PROGRAM MAIN
VAR
	rtStep						:R_Trig;
	
	rtAck						:R_Trig;
	i							:UDINT;
	fbWakeUpTmr					:TON;	
	sTime						:STRING(8);
	bAckLED						:BOOL;
	darius						:UDINT;	
	
	// Alarm	
	aErrorActive				:ARRAY[1..nNbrOfAlarms] OF WORD;
	aErrorID1					:ARRAY[1..nNbrOfAlarms] OF STRING(255);
	aErrorID2					:ARRAY[1..nNbrOfAlarms] OF STRING(255);
	afbAlarms					:ARRAY[1..nNbrOfAlarms] OF FB_TcAlarm;
	fbSource					:FB_TcSourceInfo;

	(*Vise station components*)
	rtStepViseStation			:R_Trig;

END_VAR

//InitTCPIP();
Init();
Blink();
SafetyPRG();
Alarm();
BusDiag();
Door();
Light();
Mode();
ViseProgram();
RobotCncProgram();
Robot7AxisProgram();
CNC_1();
CNC_3();
ConveyorSystem();
Mapping();

Test();
SQL_Test();


fbTime(bEnable := TRUE, dwCycle := 1);
dtSystemTime := SYSTEMTIME_TO_DT(TIMESTR:= fbTime.systemTime);
sTime := MID((SYSTEMTIME_TO_STRING(fbTime.systemTime)),8,12);

ACTION Alarm:
// Creating error acknowladge impulse
rtAck(CLK:= i_bVisePos1ErrorAckBtn OR i_bVisePos2ErrorAckBtn OR bAckHMI OR i_bErrorAckBtn_Main, Q=> bAckP);
IF rtAck.Q THEN
	afbAlarms[1].Confirm(0); afbAlarms[2].Confirm(0); afbAlarms[3].Confirm(0); afbAlarms[4].Confirm(0);
	afbAlarms[5].Confirm(0); afbAlarms[6].Confirm(0); afbAlarms[7].Confirm(0); 
	bAckHMI := FALSE;
END_IF

IF wError <> 0 OR bSafetyError_CNC45 OR ViseProgram.nState >= 200000 THEN
	bGlobalError := TRUE;
ELSE
	bGlobalError := FALSE;
END_IF

(* 
	wError.0 : Air pressure error
	wError.1 : Ethercat error
	wError.2 : 
	wError.3 : 
	wError.4 : 
	wError.5 : 
	wError.6 : 
	wError.7 : 
	wError.8 : 
	wError.9 : 
*)

aErrorActive[1].0 := wError.0;
aErrorActive[2].0 := wError.1;
aErrorActive[3].0 := i_bSafetyGroupComErr_CNC45;
aErrorActive[4].0 := i_bSafetyGroupFBErr_CNC45;
aErrorActive[5].0 := i_bSafetyGroupOtherErr_CNC45;
aErrorActive[6].0 := i_bLO1EDMErr_CNC45;
aErrorActive[7].0 := i_bLO2EDMErr_CNC45;

FOR i := 1 TO nNbrOfAlarms DO
	IF aErrorActive[i].0 THEN
		IF (afbAlarms[i].eConfirmationState <> 2 AND afbAlarms[i].nTimeCleared <> 0 AND afbAlarms[i].nTimeConfirmed <> 0) OR //Ha már volt alarm, akkor van bennük érték
			(afbAlarms[i].eConfirmationState = 1 AND afbAlarms[i].nTimeCleared = 0 AND afbAlarms[i].nTimeConfirmed = 0)	//Első futás esetén
		THEN
			IF aErrorActive[i].1 AND aErrorActive[i].2 THEN
				afbAlarms[i].ipArguments.Clear().AddString(aErrorID1[i]).AddString(aErrorID2[i]);
			ELSIF aErrorActive[i].1 THEN
				afbAlarms[i].ipArguments.Clear().AddString(aErrorID1[i]);
			ELSE
				afbAlarms[i].ipArguments.Clear();
			END_IF
			afbAlarms[i].Raise(0);
		END_IF	
	ELSE
		IF (afbAlarms[i].eConfirmationState = 2 OR afbAlarms[i].eConfirmationState = 3) AND afbAlarms[i].nTimeCleared = 0 THEN
			afbAlarms[i].Clear(0, FALSE);
		END_IF		
	END_IF
END_FOR
END_ACTION

ACTION BusDiag:
fbWakeUpTmr(IN:= NOT bFirstCycle, PT:= T#60S, Q=> , ET=> );
// eCAT network error
IF fbWakeUpTmr.Q AND (i_nBusState <> 8) THEN
	wError.1 := TRUE;	
END_IF
END_ACTION

ACTION Door:
fbDoor(
	bDoorButton:= i_bDoorRequest, 
	bOpenEnable:= TRUE (*and robot.....*),
	bEmergencyOk:= i_bLO1_CNC45,
	bWaitClose:= i_bWaitClose_CNC45,
	bDoorsClosed:= i_bDoorClosed, 
	bDoorsLocked:= i_bLO2_CNC45, 
	bBlink_1:= bBL100p100,
	bBlink_2:= bBL500p500, 
	bCloseOut=> q_bDoorLock, 
	bDoorButtonLED=> q_bDoorRequestLED,
	bCellAckLED => q_bCellAckLED, 
	bObenRequestOut=> bDoorOpenReq);
END_ACTION

ACTION Init:
IF bFirstCycle THEN
	afbAlarms[1].CreateEx(TC_Events.MyEvents.AirPE, TRUE, 0);
	afbAlarms[2].CreateEx(TC_Events.MyEvents.GenEtherCATErr, TRUE, 0);
	afbAlarms[3].CreateEx(TC_Events.MyEvents.SafetyGroupComErr, TRUE, 0);
	afbAlarms[4].CreateEx(TC_Events.MyEvents.SafetyGroupFbErr, TRUE, 0);
	afbAlarms[5].CreateEx(TC_Events.MyEvents.SafetyGroupOtherErr, TRUE, 0);
	afbAlarms[6].CreateEx(TC_Events.MyEvents.LO1EDMErr, TRUE, 0);
	afbAlarms[7].CreateEx(TC_Events.MyEvents.LO2EDMErr, TRUE, 0);
	
	fb3DCam.p_ConnectTimeout := T#2S;
	fb3DCam.p_SendTimeout := T#2S;
	fb3DCam.p_ReceiveTimeout := T#20S;
	fb3DCam.p_CloseTimeout := T#2S;
	fb3DCam.p_Name := '3D Camera';
	fb3DCam.p_RemoteHost := '192.168.81.19';
	fb3DCam.p_RemotePort := 24056;

	bFirstCycle := FALSE;
END_IF
END_ACTION

ACTION Light:
//Master on light
q_bMasterOnLED := (i_bLO1_CNC45 (*AND i_bLO2*)) OR (bBL500p500 AND 
					NOT i_bEmyStop1 AND NOT i_bEmyStop2 AND NOT i_bEmyStop3 AND
					NOT i_bEmyStop4 AND NOT i_bEmyStop5 AND NOT i_bEmyStop6);

//Error acknowledge light
bAckLED := (bGlobalError AND bBL500p500) OR 
			i_bEmyStop1 OR i_bEmyStop2 OR i_bEmyStop3 OR
			i_bEmyStop4 OR i_bEmyStop5 OR i_bEmyStop6;

q_bVise1ErrorAckLED := q_bVise2ErrorAckBtnLED := bAckLED;
	
fbNotSmartLight(
	bEmyStop:= i_bEmyStop1 OR i_bEmyStop2 OR i_bEmyStop3 OR i_bEmyStop4 OR i_bEmyStop5 OR i_bEmyStop6,
	bEmyOK:= i_bLO1_CNC45 AND i_bLO2_CNC45, 
	bError:= bGlobalError, 
	bOutOfStock:= ,
	bBuzzer := FALSE,
	bBlink := bBL500p500);
END_ACTION

ACTION Mapping:
;
END_ACTION

ACTION Mode:
// Switching mode
IF bManualModeRequest THEN
	IF (Robot7AxisProgram.nState = 0 OR Robot7AxisProgram.nState = 10000 OR Robot7AxisProgram.nState = 150000 OR Robot7AxisProgram.nState >= 200000) 
	THEN
		nMode := 2;
		bManualMode := TRUE;
		bGlobalEHA := FALSE;
	ELSE
		nMode := 1;
	END_IF
ELSE
	nMode := 0;
	bManualMode := FALSE;
	bGlobalEHA := TRUE;
END_IF

// Switching mode Vise
IF bManualModeRequestVise THEN
	IF (ViseProgram.nState = 0 OR ViseProgram.nState = 10000 OR ViseProgram.nState = 150000 OR ViseProgram.nState >= 200000) 
	THEN
		nModeVise := 2;
		bManualModeVise := TRUE;
		//bGlobalEHAVise := FALSE;
	ELSE
		nModeVise := 1;
	END_IF
ELSE
	nModeVise := 0;
	bManualModeVise := FALSE;
	//bGlobalEHAVise := TRUE;
END_IF


// Step mode for testing
rtStep(CLK:= bStepHMI OR i_bMasterOn_CNC45 OR i_bMasterOn_Main, Q=> bStepP);
IF bStepMode AND bStepP OR NOT bStepMode THEN
	bStepEnable := TRUE;
ELSE
	bStepEnable := FALSE;
END_IF

// Step mode for testing in Vise Station
rtStepViseStation(CLK:= bStepHMIViseStation OR i_bMasterOn_CNC45 OR i_bMasterOn_Main, Q=> bStepPViseStation);
IF bStepModeViseStation AND bStepPViseStation OR (NOT bStepModeViseStation) THEN
	bStepEnableViseStation := TRUE;
ELSE
	bStepEnableViseStation := FALSE;
END_IF
END_ACTION

END_PROGRAM

(* stored: Version 1.1.0.1, ProductVersion 3.1.4024.12
   POU MAIN: Id {f64088c3-f9a4-4ef8-a854-8e583a1e04fb}, SpecialFunc None
   Action Alarm: Id {74b54fed-c5dc-49fb-9aa9-6cad65b323d1}
   Action BusDiag: Id {f28fd779-3d8e-4ec9-aa56-27042a3165b6}
   Action Door: Id {6538cdd5-c667-405f-9c30-8490d92c2d68}
   Action Init: Id {d87a8829-577b-44df-8bb5-51539643ac1d}
   Action Light: Id {17fc2ff3-9ede-4c3e-bb12-242734fa3e89}
   Action Mapping: Id {35b55974-b1cc-4f74-b0f7-031aa332c171}
   Action Mode: Id {37f15e2b-fb65-4020-9798-fa6f49222fe7} *)
